TYPE SampleDataItem :
STRUCT
 	Measured : BOOL;
    Overrided : BOOL;
    Marginal : BOOL;
    FinalResults : BOOL;
END_STRUCT
END_TYPE

(* stored: Version 1.1.0.1
   DUT SampleDataItem: Id {806db45d-e7c1-4323-b4b1-30a4e6201187} *)
